// TIA Portal V17 export
TYPE "UDT_Motor"
END_TYPE
